FUNCTION_BLOCK BaseIO
VAR_INPUT
	ProcessError: BOOL;
	ProcessErrorCode: INT := 0;
END_VAR
VAR_OUTPUT
	Error: BOOL;
	ErrorCode: INT := 0;
END_VAR
VAR
	Kind: TIoKind;
END_VAR
VAR PERSISTENT
	{attribute 'TcEncoding':='UTF-8'}
	Category: STRING;
	{attribute 'TcEncoding':='UTF-8'}
	SystemName: STRING;
	{attribute 'TcEncoding':='UTF-8'}
	CustomName: STRING;
	ErrorDescription: STRING;
END_VAR

END_FUNCTION_BLOCK

(* stored: Version 1.1.0.1, ProductVersion 3.1.4024.4
   POU BaseIO: Id {bc2cc02a-bef6-49ac-bb7f-3acf66c3e4b2}, SpecialFunc None *)
